(* IEC 61131-3 sources: ICSQuartz/benchmarks/oscat_basic_find_ctrl/src, 1 file *)

(* ---- program.st ---- *)
PROGRAM PLC_PRG
VAR_INPUT
    in_pos: INT;
    in_str: STRING;
END_VAR

FIND_CTRL(in_str, in_pos);

END_PROGRAM
